TYPE stRawOutput :
STRUCT
	H1		:	BOOL;
	HEmg	:	BOOL;
	M		:	BOOL;
	Libero	:	BOOL;
END_STRUCT
END_TYPE

(* stored: Version 1.1.0.1
   DUT stRawOutput: Id {d54092bd-7ad0-0041-0dc8-150177ad10e6} *)
